TYPE SInterlock EXTENDS SConditionSpec :
STRUCT
	DefaultValue: BOOL;
END_STRUCT
END_TYPE

(* stored: Version 1.1.0.1
   DUT SInterlock: Id {852a024d-dccc-4375-8ddb-c2d32b86a0de} *)
